// TwinCAT 3 PLC project Untitled1
// ProgramVersion: 3.1.4023.0
// libraries:
//   Tc2_MC2, * (Beckhoff Automation GmbH)
//   Tc2_Standard, * (Beckhoff Automation GmbH)
//   Tc2_System, * (Beckhoff Automation GmbH)
//   Tc3_Module, * (Beckhoff Automation GmbH)
// project tree:
//   DUTs/ AirPiston.TcPOU (not stored), ClearLinkEIP.TcPOU (not stored), Homing.TcDUT, PneumaticInsertion.TcPOU (not stored), TeknicHardWire.TcPOU (not stored)
//   / PlcTask.TcTTO (not stored)
//   POUs/ DriverSequence.TcPOU, HardWireSequence.TcPOU (not stored), InsertionSequence.TcPOU, MAIN.TcPOU
//   POUs/Utility/ CEILING.TcPOU (not stored), WithinTolerance.TcPOU (not stored)
// real-time tasks:
//   TASK PlcTask: cycle T#10ms, priority 20, ADS port 350
// I/O:
//   DEVICE Device 1 (TC3 EIP Scanner), AmsNetId 5.131.216.69.2.1
//     ClearLink // <INFO> 169.254.0.152, ClearLink (ProdCode: 1, Rev: 2.93, Mac: 24:15:10:b0:30:37) </INFO> <EDS> C:\TwinCAT\3.1\Config\Io\EtherNetIP\clearlink_2.92.eds </EDS>
// variable links:
//   Untitled1/Untitled1 Instance <-> Device 1 (TC3 EIP Scanner)/ClearLink
//     PlcTask Inputs/MAIN.m0.servo.hlfb <-> Connection 1 (Input/Output)/Inputs/Motor0 HLFB Duty
//     PlcTask Inputs/MAIN.m1.servo.hlfb <-> Connection 1 (Input/Output)/Inputs/Motor1 HLFB Duty
//     PlcTask Outputs/MAIN.m0.servo.outputRegister <-> Connection 1 (Input/Output)/Outputs/Motor0 Out Reg
//     PlcTask Outputs/MAIN.m1.servo.outputRegister <-> Connection 1 (Input/Output)/Outputs/Motor1 Out Reg
//     PlcTask Outputs/MAIN.m0.servo.pulse <-> Connection 1 (Input/Output)/Outputs/Motor0 Trig Pulses
//     PlcTask Outputs/MAIN.m1.servo.pulse <-> Connection 1 (Input/Output)/Outputs/Motor1 Trig Pulses

// ---- DUTs/Homing.TcDUT
{attribute 'qualified_only'}
{attribute 'strict'}
TYPE Homing :
(
	IDLE,
	IN,
	OUT,
	OUT_FINAL,
	STOP,
	SET,
	DONE,
	
	size
);
END_TYPE

// ---- POUs/DriverSequence.TcPOU
FUNCTION_BLOCK DriverSequence
VAR_IN_OUT
	enable : BOOL;
	contUp : BOOL;
	contDown : BOOL;
	target : REAL;
END_VAR
VAR_OUTPUT
	ready : BOOL;
	
	busy : BOOL;
	position : REAL;
END_VAR
VAR
	servo : ClearLinkEIP;
	
	step : INT;
	timer : TON;
END_VAR

servo(
	bEnable:= enable,
	pulse=> , 
	outputRegister=> , 
	brakeRelease=> , 
	A=> , 
	B=> , 
	clear=> , 
	contact=> , 
	home=> , 
	outerLimit=> , 
	innerLimit=> , 
	hlfb=> , 
	homeSet=> , 
	busy=> , 
	error=> , 
	position=> , 
	targetPos=> );

IF NOT servo.homeSet THEN
	servo.homingSequence(); //homing will overwrite the bEnable input, but it must be true for homing to proceed
	RETURN;
END_IF

servo.stop();
IF contUp THEN
	servo.moveContinuous(direction := MC_Positive_Direction);
	contDown := FALSE;
END_IF

IF contDown THEN
	servo.moveContinuous(direction := MC_Negative_Direction);
	contUp := FALSE;
END_IF


IF target >= 0 THEN
	servo.moveAbsolute(newTarget := target);
	//target := 0;
END_IF


IF servo.innerLimit THEN
	contDown := FALSE;
END_IF
IF servo.home THEN
	contUp := FALSE;
END_IF

position := servo.position;
busy := servo.busy;

METHOD autoSequence : BOOL
VAR_INPUT
END_VAR
timer(IN:= , PT:= , Q=> , ET=> );

CASE step OF
	0: //+continuous for 5s
		timer.IN := TRUE;
		timer.PT := T#5S;
		
		contUp := TRUE;
		
		IF timer.Q THEN
			timer.IN := FALSE;
			contUp := FALSE;
			step := 10;
		END_IF
		
	10: //target
		IF position = 150 AND NOT busy THEN
			target := -1;
			step := 20;
			RETURN;
		END_IF
		
		target := 150;
		
		IF busy THEN
			//step := 11;
		END_IF
		
	11:
		//paste top part of 10 if does not work
	
	20: //-continuous 2s
		timer.IN := TRUE;
		timer.PT := T#2S;
		
		contDown := TRUE;
		
		IF timer.Q THEN
			timer.IN := FALSE;
			contDown := FALSE;
			step := 30;
		END_IF
	
	
	30: //target 0
		target := 0;
		
		IF busy THEN
			step := 31;
		END_IF
		
	31:
		IF position = 0 AND NOT busy THEN
			target := -1;
			step := 40;
			RETURN;
		END_IF
		
	40:
		timer.IN := TRUE;
		timer.PT := T#1S;
		
		IF timer.Q THEN
			timer.IN := FALSE;
			step := 0;
		END_IF
END_CASE
END_METHOD

END_FUNCTION_BLOCK

// ---- POUs/InsertionSequence.TcPOU
FUNCTION_BLOCK InsertionSequence
VAR_IN_OUT
	
END_VAR
VAR
	insertion : PneumaticInsertion;
	
	contUp, contDown : BOOL;
	vTarget : REAL := -1;
	press, release : BOOL;
END_VAR

insertion(
	enable:= TRUE, 
	slider=> , 
	screw=> , 
	contact=> , 
	home=> , 
	ready=> , 
	busy=> , 
	error=> , 
	homeSet=> );

IF NOT insertion.homeSet THEN
	insertion.homingSequence();
	RETURN;
END_IF

insertion.stop(); //executes if any of the following are false

IF contUp THEN
	insertion.slideContinuous(direction := MC_Positive_Direction);
	contDown := FALSE;
END_IF

IF contDown THEN
	insertion.slideContinuous(direction := MC_Negative_Direction);
	contUp := FALSE;
END_IF

IF vTarget >= 0 THEN
	insertion.slideAbsolute(targetPos := vTarget);
END_IF

END_FUNCTION_BLOCK

// ---- POUs/MAIN.TcPOU
PROGRAM MAIN
VAR
	m0 : DriverSequence();
	m1 : DriverSequence();
	
	enable : BOOL := TRUE;
	
	ready : BOOL;
	contUp : BOOL;
	contDown : BOOL;
	target : REAL := -1;
	
	auto : BOOL := TRUE;
	
	step : INT;
	timer : TON;
END_VAR

IF m0.ready AND m1.ready AND auto THEN
	autoSequence();
END_IF

m0(
	enable:= enable,
	contUp:= contUp, 
	contDown:= contDown, 
	target:= target,
	ready=> );

m1(
	enable:= enable,
	contUp:= contUp, 
	contDown:= contDown, 
	target:= target,
	ready=> );
	
(*
this module contains 2 ClearLink MC Motors
motors can be controlled manually or with an automatic demo routine
motors must be enabled and homed before use

contUp - continuous positive direction
contDown - continuous negative direction

target - target a specified position >= 0
*)

METHOD autoSequence : BOOL
VAR_INPUT
END_VAR
timer(IN:= , PT:= , Q=> , ET=> );

CASE step OF
	0: //+continuous for 5s
		timer.IN := TRUE;
		timer.PT := T#5S;
		
		contUp := TRUE;
		
		IF timer.Q THEN
			timer.IN := FALSE;
			contUp := FALSE;
			step := 10;
		END_IF
		
	10: //target
		IF m0.position = 150 AND NOT m0.busy AND m1.position = 150 AND NOT m1.busy THEN
			target := -1;
			step := 20;
			RETURN;
		END_IF
		
		target := 150;
		
		IF m0.busy AND m1.busy THEN
			//step := 11;
		END_IF
		
	11:
		//
	
	20: //-continuous 2s
		timer.IN := TRUE;
		timer.PT := T#2S;
		
		contDown := TRUE;
		
		IF timer.Q THEN
			timer.IN := FALSE;
			contDown := FALSE;
			step := 30;
		END_IF
	
	
	30: //target 0
		target := 0;
		
		IF m0.busy AND m1.busy THEN
			step := 31;
		END_IF
		
	31:
		IF m0.position = 0 AND NOT m0.busy AND m1.position = 0 AND NOT m1.busy THEN
			target := -1;
			step := 40;
			RETURN;
		END_IF
		
	40:
		timer.IN := TRUE;
		timer.PT := T#1S;
		
		IF timer.Q THEN
			timer.IN := FALSE;
			step := 0;
		END_IF
END_CASE
END_METHOD

END_PROGRAM
